(* IEC 61131-3 sources: automationbase/examples, 6 files *)

(* ---- ResetCommandExample.st ---- *)
NAMESPACE Simatic.Ax.AutomationBase.Examples

    USING Simatic.Ax.AutomationBase;
    USING Simatic.Ax.IO.Input;

    /// Example demonstrating centralized reset command management
    /// Shows how to use ResetCommandManager with automatic edge detection and IBinSignal

    /// Example equipment with custom reset logic
    CLASS ExampleEquipmentWithCustomReset EXTENDS EquipmentBase
        VAR PUBLIC
            Running : BOOL;
            ErrorCondition : BOOL;  // Simulated error condition
            ResetCounter : INT;     // Tracks number of resets
        END_VAR

        METHOD PROTECTED OVERRIDE InitUser
            Running := FALSE;
            ResetCounter := 0;
        END_METHOD

        METHOD PROTECTED OVERRIDE RunCyclicUserCode
            // Simulate error condition
            IF (ErrorCondition AND NOT THIS.HasError()) THEN
                THIS.SetError(errorState := ErrorState#OtherError,
                             errorText := 'Simulated error');
            END_IF;

            // Normal operation when no error
            IF (NOT THIS.HasError()) THEN
                IF (THIS.GetStartupStatus() = StartUpStatus#AutoStartedUp) THEN
                    Running := TRUE;
                ELSE
                    Running := FALSE;
                END_IF;
            ELSE
                Running := FALSE;
            END_IF;
        END_METHOD

        /// Custom reset logic - override to add equipment-specific reset behavior
        METHOD PROTECTED OVERRIDE ResetFaultUser
            // Call base implementation to clear error
            SUPER^.ResetFaultUser();

            // Add custom reset logic
            ResetCounter := ResetCounter + 1;
            Running := FALSE;

            // Clear error condition
            ErrorCondition := FALSE;

            // Could add more equipment-specific reset actions:
            // - Reset internal state machines
            // - Clear buffers
            // - Reset actuators to safe position
            // - Log reset event
        END_METHOD
    END_CLASS

    /// Example equipment with different custom reset logic
    CLASS ExampleMotorWithReset EXTENDS EquipmentBase
        VAR PUBLIC
            Speed : REAL;
            Position : REAL;
            ErrorCondition : BOOL;
        END_VAR

        METHOD PROTECTED OVERRIDE InitUser
            Speed := 0.0;
            Position := 0.0;
        END_METHOD

        METHOD PROTECTED OVERRIDE RunCyclicUserCode
            IF (ErrorCondition AND NOT THIS.HasError()) THEN
                THIS.SetError(errorState := ErrorState#OtherError,
                             errorText := 'Motor error');
            END_IF;

            IF (NOT THIS.HasError()) THEN
                IF (THIS.GetStartupStatus() = StartUpStatus#AutoStartedUp) THEN
                    Speed := 100.0;
                END_IF;
            ELSE
                Speed := 0.0;
            END_IF;
        END_METHOD

        /// Motor-specific reset logic
        METHOD PROTECTED OVERRIDE ResetFaultUser
            // Call base implementation
            SUPER^.ResetFaultUser();

            // Motor-specific reset
            Speed := 0.0;
            ErrorCondition := FALSE;
            // Position is NOT reset - we keep position information
        END_METHOD
    END_CLASS

    /// Example program showing centralized reset with automatic edge detection
    PROGRAM ResetCommandExample
        VAR
            // Equipment instances
            equipment1 : ExampleEquipmentWithCustomReset;
            equipment2 : ExampleEquipmentWithCustomReset;
            motor1 : ExampleMotorWithReset;

            // Shared infrastructure
            modeManager : OperatingModeManager;
            resetManager : ResetCommandManager;  // Central reset manager

            // Reset signal (connected to HMI button)
            resetButtonSignal : BinSignal;

            // Control inputs
            simulateError1 : BOOL;
            simulateError2 : BOOL;
            simulateError3 : BOOL;

            // Monitoring outputs
            hmi_ResetActive : BOOL;
            hmi_AnyError : BOOL;
        END_VAR

        // ============================================
        // CONFIGURATION (once during initialization)
        // ============================================

        // Configure equipment 1
        equipment1.Mode := modeManager;
        equipment1.ResetCommand := resetManager;  // Connect to central reset
        equipment1.ErrorCondition := simulateError1;

        // Configure equipment 2
        equipment2.Mode := modeManager;
        equipment2.ResetCommand := resetManager;  // Same reset manager
        equipment2.ErrorCondition := simulateError2;

        // Configure motor
        motor1.Mode := modeManager;
        motor1.ResetCommand := resetManager;  // Same reset manager
        motor1.ErrorCondition := simulateError3;

        // Connect reset signal to manager
        resetManager.ResetSignal := resetButtonSignal;

        // ============================================
        // SIGNAL INPUT
        // ============================================

        // Read reset button signal (connect to your HMI button input)
        resetButtonSignal.ReadCyclic(signal := (* your HMI reset button input *), valid := TRUE);

        // ============================================
        // CYCLIC EXECUTION
        // ============================================

        // All equipment will automatically:
        // - Report errors via ReportError() when HasError() is TRUE
        // - Check for reset command via GetResetCommand()
        // - Call ResetFaultUser() when reset is active and equipment has error
        equipment1.RunCyclic();
        equipment2.RunCyclic();
        motor1.RunCyclic();

        // IMPORTANT: ResetManager must run after all equipment
        // RunCyclic() automatically:
        // - Detects reset signal rising edge via ResetSignal.QRis()
        // - Activates reset command for exactly one cycle
        // - Clears error flag on reset
        resetManager.RunCyclic();

        // ============================================
        // MONITORING
        // ============================================

        // Check if any equipment has reported errors
        hmi_AnyError := resetManager.AnyErrorActive();

        // Check if reset command is currently active
        hmi_ResetActive := resetManager.IsResetActive();

        // Example flow:
        // 1. Equipment has error → AnyErrorActive() = TRUE
        // 2. Reset button pressed (rising edge) → IsResetActive() = TRUE for one cycle
        // 3. Equipment resets → AnyErrorActive() = FALSE
        // 4. Next cycle → IsResetActive() = FALSE
    END_PROGRAM

END_NAMESPACE

(* ---- AxisSupervisionExample.st ---- *)
USING Simatic.Ax.AutomationBase;

NAMESPACE Examples

    /// Beispielprogramm für die Verwendung der AxisSupervision Klasse
    PROGRAM AxisSupervisionExample
        VAR
            // Achsenüberwachung Instanz
            axis_supervision : AxisSupervision;

            // Simulierte Achsendaten
            axis_current_pos : REAL;      // Aktuelle Position der Achse
            axis_target_pos : REAL;       // Zielposition
            axis_start_pos : REAL;        // Startposition

            // Steuerungsvariablen
            start_movement : BOOL;        // Trigger zum Starten der Bewegung
            reset_error : BOOL;           // Trigger zum Zurücksetzen von Fehlern

            // Statusvariablen
            movement_active : BOOL;
            error_occurred : BOOL;
            error_code : SupervisionError;

            // Simulationsvariablen
            simulate_movement : BOOL := TRUE;
            movement_speed : REAL;        // Geschwindigkeit der simulierten Bewegung
        END_VAR

        //=============================================================================
        // INITIALISIERUNG (einmalig beim Start)
        //=============================================================================

        // Konfiguration der Überwachungsparameter
        axis_supervision.t_action := T#3s;      // 3 Sekunden bis Startposition verlassen werden muss
        axis_supervision.t_reaction := T#10s;   // 10 Sekunden bis Zielposition erreicht werden muss
        axis_supervision.tolerance := REAL#0.5; // Toleranz von 0.5 Einheiten

        //=============================================================================
        // ZYKLISCHE AUSFÜHRUNG
        //=============================================================================

        // Positionen an Überwachung übergeben
        axis_supervision.current_position := axis_current_pos;
        axis_supervision.start_position := axis_start_pos;
        axis_supervision.target_position := axis_target_pos;

        // Bewegung starten
        IF start_movement AND NOT movement_active THEN
            // Setze Startposition auf aktuelle Position
            axis_start_pos := axis_current_pos;

            // Starte Überwachung
            axis_supervision.StartSupervision();
            movement_active := TRUE;
            start_movement := FALSE;
        END_IF;

        // Überwachung ausführen (muss zyklisch aufgerufen werden)
        axis_supervision.Execute();

        // Bewegungssimulation (in echter Anwendung durch echte Achsensteuerung ersetzen)
        IF simulate_movement AND movement_active THEN
            THIS.SimulateAxisMovement();
        END_IF;

        // Status auslesen
        error_occurred := axis_supervision.HasError();
        error_code := axis_supervision.GetError();

        // Fehlerbehandlung
        IF error_occurred THEN
            movement_active := FALSE;

            // Fehlerausgabe
            CASE error_code OF
                SupervisionError#ERROR_ACTION_TIMEOUT:
                    // Fehler: Achse hat Startposition nicht rechtzeitig verlassen
                    // Hier könnte z.B. eine Alarmmeldung ausgegeben werden
                    ;

                SupervisionError#ERROR_REACTION_TIMEOUT:
                    // Fehler: Achse hat Zielposition nicht rechtzeitig erreicht
                    // Hier könnte z.B. eine Alarmmeldung ausgegeben werden
                    ;
            END_CASE;
        END_IF;

        // Fehler zurücksetzen
        IF reset_error THEN
            axis_supervision.ResetError();
            error_occurred := FALSE;
            error_code := SupervisionError#NO_ERROR;
            reset_error := FALSE;
        END_IF;

        // Bewegung erfolgreich abgeschlossen
        IF axis_supervision.HasReachedTarget() THEN
            movement_active := FALSE;
        END_IF;

    END_PROGRAM

    /// Simuliert eine Achsenbewegung (nur für Demonstrationszwecke)
    METHOD PRIVATE SimulateAxisMovement
        VAR_TEMP
            distance_to_target : REAL;
            direction : REAL;
        END_VAR

        // Berechne Distanz und Richtung zum Ziel
        distance_to_target := axis_target_pos - axis_current_pos;

        IF Abs(distance_to_target) > axis_supervision.tolerance THEN
            // Bestimme Bewegungsrichtung
            IF distance_to_target > REAL#0.0 THEN
                direction := REAL#1.0;
            ELSE
                direction := REAL#-1.0;
            END_IF;

            // Bewege Achse (Geschwindigkeit: 1.0 Einheiten pro Zyklus)
            movement_speed := REAL#1.0;
            axis_current_pos := axis_current_pos + (direction * movement_speed);
        END_IF;
    END_METHOD

END_NAMESPACE

(* ---- LoggingExample.st ---- *)
USING Simatic.Ax.AutomationBase;

NAMESPACE Examples

    /// Example program demonstrating the logging functionality
    PROGRAM LoggingExample
        VAR
            // Logger instances
            ringLogger : RingBufferLogger;
            consoleLogger : ConsoleLogger;

            // Buffer for ring buffer logger (100 entries)
            logBuffer : ARRAY[0..99] OF LogEntry;

            // Example variables
            temperature : REAL := 25.0;
            pressure : REAL := 1.0;
            errorOccurred : BOOL := FALSE;
            cycleCount : DINT := 0;
        END_VAR

        // Initialize loggers (call once at startup)
        ringLogger.Buffer := REF(logBuffer);
        ringLogger.MinLogLevel := LogLevel#Info;  // Log Info and above

        consoleLogger.Enabled := TRUE;
        consoleLogger.MinLogLevel := LogLevel#Debug;  // Log everything

        // Increment cycle counter
        cycleCount := cycleCount + 1;

        //=============================================================================
        // EXAMPLE 1: Simple logging
        //=============================================================================
        IF (cycleCount = 1) THEN
            ringLogger.LogInfo('System started');
            consoleLogger.LogInfo('System started');
        END_IF;

        //=============================================================================
        // EXAMPLE 2: Conditional logging based on values
        //=============================================================================
        IF (temperature > 80.0) THEN
            ringLogger.LogWarning('Temperature high: 85.5 degC');
        END_IF;

        IF (temperature > 100.0) THEN
            ringLogger.LogError('Temperature critical: 105.0 degC');
        END_IF;

        //=============================================================================
        // EXAMPLE 3: Logging with source information
        //=============================================================================
        IF (pressure < 0.5) THEN
            ringLogger.LogWithSource(
                level := LogLevel#Warning,
                message := 'Pressure low',
                source := 'PressureSensor1'
            );
        END_IF;

        //=============================================================================
        // EXAMPLE 4: Debug logging
        //=============================================================================
        IF (cycleCount MOD 1000 = 0) THEN
            consoleLogger.LogDebug('Cycle 1000 reached');
        END_IF;

        //=============================================================================
        // EXAMPLE 5: Checking log statistics
        //=============================================================================
        IF ringLogger.HasLevel(LogLevel#Error) THEN
            // React to errors in log
            errorOccurred := TRUE;
        END_IF;

        //=============================================================================
        // EXAMPLE 6: Reading log entries
        //=============================================================================
        VAR
            entry : LogEntry;
            valid : BOOL;
            i : DINT;
        END_VAR

        // Read last 5 entries
        FOR i := 0 TO 4 DO
            IF (i < ringLogger.GetCount()) THEN
                ringLogger.GetEntryAt(
                    index := ringLogger.GetCount() - 1 - i,
                    entry => entry,
                    valid => valid
                );

                IF valid THEN
                    // Process entry
                    CASE entry.Level OF
                        LogLevel#Error:
                            // Handle error entry
                            ;
                        LogLevel#Warning:
                            // Handle warning entry
                            ;
                    END_CASE;
                END_IF;
            END_IF;
        END_FOR;

        //=============================================================================
        // EXAMPLE 7: Log statistics
        //=============================================================================
        VAR
            totalLogs : DINT;
            errorCount : DINT;
            warningCount : DINT;
            infoCount : DINT;
        END_VAR

        totalLogs := ringLogger.GetCount();
        errorCount := ringLogger.GetErrorCount();
        warningCount := ringLogger.GetWarningCount();
        infoCount := ringLogger.GetInfoCount();

        //=============================================================================
        // EXAMPLE 8: Clearing logs
        //=============================================================================
        VAR
            clearLogs : BOOL := FALSE;
        END_VAR

        IF clearLogs THEN
            ringLogger.Clear();
            consoleLogger.Clear();
            clearLogs := FALSE;
        END_IF;

    END_PROGRAM

END_NAMESPACE

(* ---- PneumaticCylinderExample.st ---- *)
USING Simatic.Ax.AutomationBase;

NAMESPACE Examples

    /// Beispielprogramm für die Verwendung der AxisSupervision Klasse
    /// Zeigt die Überwachung eines Pneumatikzylinders mit Endschaltern
    PROGRAM PneumaticCylinderSupervisionExample
        VAR
            // Achsenüberwachung Instanz
            cylinder_supervision : AxisSupervision;

            // Pneumatikzylinder Steuerung
            cylinder_extend : BOOL;           // Ausfahren-Signal
            cylinder_retract : BOOL;          // Einfahren-Signal

            // Endschalter (Sensoren)
            sensor_retracted : BOOL;          // Endschalter: Zylinder eingefahren
            sensor_extended : BOOL;           // Endschalter: Zylinder ausgefahren

            // Steuerungsvariablen
            start_extend : BOOL;              // Trigger zum Ausfahren
            start_retract : BOOL;             // Trigger zum Einfahren
            reset_error : BOOL;               // Trigger zum Zurücksetzen von Fehlern

            // Statusvariablen
            movement_active : BOOL;
            error_occurred : BOOL;
            error_code : SupervisionError;
            cylinder_state : CylinderState;
        END_VAR

        //=============================================================================
        // INITIALISIERUNG (einmalig beim Start)
        //=============================================================================

        // Konfiguration der Überwachungsparameter
        cylinder_supervision.t_action := T#2s;      // 2 Sekunden bis Bewegung beginnt
        cylinder_supervision.t_reaction := T#5s;    // 5 Sekunden bis Endposition erreicht

        //=============================================================================
        // ZYKLISCHE AUSFÜHRUNG
        //=============================================================================

        // Ausfahren starten
        IF start_extend AND NOT movement_active AND NOT error_occurred THEN
            IF sensor_retracted THEN  // Nur ausfahren, wenn eingefahren
                cylinder_extend := TRUE;
                cylinder_retract := FALSE;

                // Überwachung konfigurieren und starten
                // has_left_start = TRUE, wenn Zylinder nicht mehr eingefahren ist
                // has_reached_target = TRUE, wenn Zylinder ausgefahren ist
                cylinder_supervision.StartSupervision();
                movement_active := TRUE;
                cylinder_state := CylinderState#Extending;
            END_IF;
            start_extend := FALSE;
        END_IF;

        // Einfahren starten
        IF start_retract AND NOT movement_active AND NOT error_occurred THEN
            IF sensor_extended THEN  // Nur einfahren, wenn ausgefahren
                cylinder_extend := FALSE;
                cylinder_retract := TRUE;

                // Überwachung konfigurieren und starten
                cylinder_supervision.StartSupervision();
                movement_active := TRUE;
                cylinder_state := CylinderState#Retracting;
            END_IF;
            start_retract := FALSE;
        END_IF;

        // Signale für Überwachung setzen (abhängig von Bewegungsrichtung)
        CASE cylinder_state OF
            CylinderState#Extending:
                // Beim Ausfahren:
                // - Startposition verlassen = Sensor "eingefahren" nicht mehr aktiv
                // - Zielposition erreicht = Sensor "ausgefahren" aktiv
                cylinder_supervision.has_left_start := NOT sensor_retracted;
                cylinder_supervision.has_reached_target := sensor_extended;

            CylinderState#Retracting:
                // Beim Einfahren:
                // - Startposition verlassen = Sensor "ausgefahren" nicht mehr aktiv
                // - Zielposition erreicht = Sensor "eingefahren" aktiv
                cylinder_supervision.has_left_start := NOT sensor_extended;
                cylinder_supervision.has_reached_target := sensor_retracted;

            CylinderState#Idle:
                cylinder_supervision.has_left_start := FALSE;
                cylinder_supervision.has_reached_target := FALSE;
        END_CASE;

        // Überwachung ausführen (muss zyklisch aufgerufen werden)
        cylinder_supervision.Execute();

        // Status auslesen
        error_occurred := cylinder_supervision.HasError();
        error_code := cylinder_supervision.GetError();

        // Fehlerbehandlung
        IF error_occurred THEN
            // Zylinder stoppen
            cylinder_extend := FALSE;
            cylinder_retract := FALSE;
            movement_active := FALSE;
            cylinder_state := CylinderState#Error;

            // Fehlerausgabe
            CASE error_code OF
                SupervisionError#ERROR_ACTION_TIMEOUT:
                    // Fehler: Zylinder hat Startposition nicht rechtzeitig verlassen
                    // Mögliche Ursachen:
                    // - Ventil defekt
                    // - Zylinder blockiert
                    // - Sensor defekt
                    ;

                SupervisionError#ERROR_REACTION_TIMEOUT:
                    // Fehler: Zylinder hat Zielposition nicht rechtzeitig erreicht
                    // Mögliche Ursachen:
                    // - Zylinder zu langsam
                    // - Mechanische Blockierung
                    // - Sensor defekt
                    // - Druckluft zu niedrig
                    ;
            END_CASE;
        END_IF;

        // Fehler zurücksetzen
        IF reset_error THEN
            cylinder_supervision.ResetError();
            error_occurred := FALSE;
            error_code := SupervisionError#NO_ERROR;
            cylinder_state := CylinderState#Idle;
            reset_error := FALSE;
        END_IF;

        // Bewegung erfolgreich abgeschlossen
        IF cylinder_supervision.HasReachedTarget() AND movement_active THEN
            cylinder_extend := FALSE;
            cylinder_retract := FALSE;
            movement_active := FALSE;
            cylinder_state := CylinderState#Idle;
        END_IF;

    END_PROGRAM

    /// Zustände des Pneumatikzylinders
    TYPE
        CylinderState : INT (
            Idle := 0,          // Ruhezustand
            Extending := 1,     // Ausfahren
            Retracting := 2,    // Einfahren
            Error := 99         // Fehlerzustand
        ) := Idle;
    END_TYPE

END_NAMESPACE

(* ---- ServoAxisExample.st ---- *)
USING Simatic.Ax.AutomationBase;

NAMESPACE Examples

    /// Beispielprogramm für die Verwendung der AxisSupervision Klasse
    /// Zeigt die Überwachung einer Servo-Achse mit Positionsrückmeldung
    PROGRAM ServoAxisSupervisionExample
        VAR
            // Achsenüberwachung Instanz
            axis_supervision : AxisSupervision;

            // Servo-Achse Daten
            axis_actual_position : REAL;      // Aktuelle Position der Achse
            axis_target_position : REAL;      // Zielposition
            axis_start_position : REAL;       // Startposition bei Bewegungsbeginn
            axis_tolerance : REAL := REAL#1.0; // Toleranz für "Position erreicht"

            // Steuerungsvariablen
            start_movement : BOOL;            // Trigger zum Starten der Bewegung
            reset_error : BOOL;               // Trigger zum Zurücksetzen von Fehlern

            // Statusvariablen
            movement_active : BOOL;
            error_occurred : BOOL;
            error_code : SupervisionError;
        END_VAR

        //=============================================================================
        // INITIALISIERUNG (einmalig beim Start)
        //=============================================================================

        // Konfiguration der Überwachungsparameter
        axis_supervision.t_action := T#1s;      // 1 Sekunde bis Achse beginnt sich zu bewegen
        axis_supervision.t_reaction := T#10s;   // 10 Sekunden bis Zielposition erreicht

        //=============================================================================
        // ZYKLISCHE AUSFÜHRUNG
        //=============================================================================

        // Bewegung starten
        IF start_movement AND NOT movement_active AND NOT error_occurred THEN
            // Startposition merken
            axis_start_position := axis_actual_position;

            // Überwachung starten
            axis_supervision.StartSupervision();
            movement_active := TRUE;
            start_movement := FALSE;

            // Hier würde die Achse den Fahrbefehl zur Zielposition erhalten
            // z.B. axis_controller.MoveAbsolute(axis_target_position);
        END_IF;

        // Signale für Überwachung berechnen
        IF movement_active THEN
            // Hat Achse Startposition verlassen? (außerhalb Toleranz)
            axis_supervision.has_left_start :=
                (Abs(axis_actual_position - axis_start_position) > axis_tolerance);

            // Hat Achse Zielposition erreicht? (innerhalb Toleranz)
            axis_supervision.has_reached_target :=
                (Abs(axis_actual_position - axis_target_position) <= axis_tolerance);
        ELSE
            axis_supervision.has_left_start := FALSE;
            axis_supervision.has_reached_target := FALSE;
        END_IF;

        // Überwachung ausführen (muss zyklisch aufgerufen werden)
        axis_supervision.Execute();

        // Status auslesen
        error_occurred := axis_supervision.HasError();
        error_code := axis_supervision.GetError();

        // Fehlerbehandlung
        IF error_occurred THEN
            movement_active := FALSE;

            // Hier würde die Achse gestoppt werden
            // z.B. axis_controller.Stop();

            // Fehlerausgabe
            CASE error_code OF
                SupervisionError#ERROR_ACTION_TIMEOUT:
                    // Fehler: Achse hat nicht begonnen sich zu bewegen
                    // Mögliche Ursachen:
                    // - Achse nicht freigegeben
                    // - Antrieb im Fehler
                    // - Mechanische Blockierung
                    ;

                SupervisionError#ERROR_REACTION_TIMEOUT:
                    // Fehler: Achse hat Zielposition nicht rechtzeitig erreicht
                    // Mögliche Ursachen:
                    // - Achse zu langsam parametriert
                    // - Mechanische Blockierung
                    // - Last zu groß
                    ;
            END_CASE;
        END_IF;

        // Fehler zurücksetzen
        IF reset_error THEN
            axis_supervision.ResetError();
            error_occurred := FALSE;
            error_code := SupervisionError#NO_ERROR;
            reset_error := FALSE;
        END_IF;

        // Bewegung erfolgreich abgeschlossen
        IF axis_supervision.HasReachedTarget() AND movement_active THEN
            movement_active := FALSE;
        END_IF;

    END_PROGRAM

    /// Hilfsfunktion für Absolutwert (falls System.Math nicht verfügbar)
    METHOD PRIVATE Abs : REAL
        VAR_INPUT
            value : REAL;
        END_VAR

        IF value < REAL#0.0 THEN
            Abs := -value;
        ELSE
            Abs := value;
        END_IF;
    END_METHOD

END_NAMESPACE

(* ---- SupervisionExample.st ---- *)
USING Simatic.Ax.AutomationBase;

NAMESPACE Examples

    /// Universelles Beispielprogramm für die Verwendung der Supervision Klasse
    /// Zeigt verschiedene Anwendungsfälle der generischen Überwachung
    PROGRAM SupervisionExample
        VAR
            //=============================================================================
            // Beispiel 1: Pneumatikzylinder ausfahren
            //=============================================================================
            supervision_cylinder_extend : Supervision;
            cylinder_extend_valve : BOOL;           // Ventil zum Ausfahren
            cylinder_sensor_extended : BOOL;        // Sensor: Zylinder ausgefahren
            start_cylinder_extend : BOOL;           // Trigger

            //=============================================================================
            // Beispiel 2: Motor starten
            //=============================================================================
            supervision_motor_start : Supervision;
            motor_start_command : BOOL;             // Startbefehl für Motor
            motor_running_feedback : BOOL;          // Rückmeldung: Motor läuft
            start_motor : BOOL;                     // Trigger

            //=============================================================================
            // Beispiel 3: Ventil schließen
            //=============================================================================
            supervision_valve_close : Supervision;
            valve_close_command : BOOL;             // Befehl zum Schließen
            valve_closed_sensor : BOOL;             // Sensor: Ventil geschlossen
            close_valve : BOOL;                     // Trigger

            //=============================================================================
            // Beispiel 4: Sensor-Überwachung (Signal soll inaktiv werden)
            //=============================================================================
            supervision_sensor_clear : Supervision;
            sensor_signal : BOOL;                   // Zu überwachender Sensor
            wait_for_sensor_clear : BOOL;           // Trigger

            //=============================================================================
            // Beispiel 5: Zweistufige Überwachung (Aktion + Reaktion)
            //=============================================================================
            supervision_action : Supervision;       // Überwacht: Bewegung beginnt
            supervision_reaction : Supervision;     // Überwacht: Bewegung endet
            actuator_command : BOOL;                // Befehl an Aktuator
            actuator_start_sensor : BOOL;           // Sensor: Startposition verlassen
            actuator_target_sensor : BOOL;          // Sensor: Zielposition erreicht
            start_actuator : BOOL;                  // Trigger

            // Gemeinsame Variablen
            reset_errors : BOOL;                    // Reset für alle Fehler
        END_VAR

        //=============================================================================
        // BEISPIEL 1: PNEUMATIKZYLINDER AUSFAHREN
        // Überwacht, ob Sensor "ausgefahren" innerhalb von 5 Sekunden aktiv wird
        //=============================================================================

        // Konfiguration (einmalig)
        supervision_cylinder_extend.timeout := T#5s;
        supervision_cylinder_extend.behavior := SupervisionBehavior#Action;  // Signal soll TRUE werden

        // Bewegung starten
        IF start_cylinder_extend THEN
            cylinder_extend_valve := TRUE;
            supervision_cylinder_extend.Start();
            start_cylinder_extend := FALSE;
        END_IF;

        // Zyklisch: Signal übergeben und überwachen
        supervision_cylinder_extend.Execute(signal := cylinder_sensor_extended);

        // Fehlerbehandlung
        IF supervision_cylinder_extend.HasError() THEN
            cylinder_extend_valve := FALSE;
            // Fehler: Zylinder hat Endposition nicht erreicht
        END_IF;

        // Erfolgreich abgeschlossen
        IF supervision_cylinder_extend.IsCompleted() THEN
            // Zylinder ist ausgefahren
        END_IF;

        //=============================================================================
        // BEISPIEL 2: MOTOR STARTEN
        // Überwacht, ob Motor-Rückmeldung innerhalb von 3 Sekunden aktiv wird
        //=============================================================================

        // Konfiguration
        supervision_motor_start.timeout := T#3s;
        supervision_motor_start.behavior := SupervisionBehavior#Action;

        // Motor starten
        IF start_motor THEN
            motor_start_command := TRUE;
            supervision_motor_start.Start();
            start_motor := FALSE;
        END_IF;

        // Zyklisch überwachen
        supervision_motor_start.Execute(signal := motor_running_feedback);

        IF supervision_motor_start.HasError() THEN
            motor_start_command := FALSE;
            // Fehler: Motor hat nicht gestartet
        END_IF;

        //=============================================================================
        // BEISPIEL 3: VENTIL SCHLIESSEN
        // Überwacht, ob Ventil innerhalb von 2 Sekunden geschlossen ist
        //=============================================================================

        // Konfiguration
        supervision_valve_close.timeout := T#2s;
        supervision_valve_close.behavior := SupervisionBehavior#Action;

        // Ventil schließen
        IF close_valve THEN
            valve_close_command := TRUE;
            supervision_valve_close.Start();
            close_valve := FALSE;
        END_IF;

        // Zyklisch überwachen
        supervision_valve_close.Execute(signal := valve_closed_sensor);

        IF supervision_valve_close.HasError() THEN
            // Fehler: Ventil hat nicht geschlossen
        END_IF;

        //=============================================================================
        // BEISPIEL 4: SENSOR-ÜBERWACHUNG (Signal soll inaktiv werden)
        // Überwacht, ob Sensor innerhalb von 10 Sekunden inaktiv wird
        //=============================================================================

        // Konfiguration
        supervision_sensor_clear.timeout := T#10s;
        supervision_sensor_clear.behavior := SupervisionBehavior#Reaction;  // Signal soll FALSE werden

        // Überwachung starten
        IF wait_for_sensor_clear THEN
            supervision_sensor_clear.Start();
            wait_for_sensor_clear := FALSE;
        END_IF;

        // Zyklisch überwachen
        supervision_sensor_clear.Execute(signal := sensor_signal);

        IF supervision_sensor_clear.HasError() THEN
            // Fehler: Sensor ist nicht inaktiv geworden
        END_IF;

        //=============================================================================
        // BEISPIEL 5: ZWEISTUFIGE ÜBERWACHUNG (Aktion + Reaktion)
        // Überwacht erst, ob Bewegung beginnt, dann ob sie endet
        //=============================================================================

        // Konfiguration
        supervision_action.timeout := T#2s;
        supervision_action.behavior := SupervisionBehavior#Action;      // Startposition verlassen
        supervision_reaction.timeout := T#10s;
        supervision_reaction.behavior := SupervisionBehavior#Action;    // Zielposition erreichen

        // Bewegung starten
        IF start_actuator THEN
            actuator_command := TRUE;
            supervision_action.Start();
            start_actuator := FALSE;
        END_IF;

        // Phase 1: Aktionsüberwachung (Bewegung beginnt)
        IF supervision_action.IsActive() THEN
            supervision_action.Execute(signal := actuator_start_sensor);

            // Wenn Startposition verlassen, starte Reaktionsüberwachung
            IF supervision_action.IsCompleted() THEN
                supervision_reaction.Start();
            END_IF;

            IF supervision_action.HasError() THEN
                actuator_command := FALSE;
                // Fehler: Bewegung hat nicht begonnen
            END_IF;
        END_IF;

        // Phase 2: Reaktionsüberwachung (Bewegung endet)
        IF supervision_reaction.IsActive() THEN
            supervision_reaction.Execute(signal := actuator_target_sensor);

            IF supervision_reaction.IsCompleted() THEN
                actuator_command := FALSE;
                // Erfolgreich: Zielposition erreicht
            END_IF;

            IF supervision_reaction.HasError() THEN
                actuator_command := FALSE;
                // Fehler: Zielposition nicht erreicht
            END_IF;
        END_IF;

        //=============================================================================
        // GEMEINSAME FEHLERBEHANDLUNG
        //=============================================================================

        // Alle Fehler zurücksetzen
        IF reset_errors THEN
            supervision_cylinder_extend.Reset();
            supervision_motor_start.Reset();
            supervision_valve_close.Reset();
            supervision_sensor_clear.Reset();
            supervision_action.Reset();
            supervision_reaction.Reset();
            reset_errors := FALSE;
        END_IF;

    END_PROGRAM

END_NAMESPACE
